// TIA Portal project "ProfiZumo" (V17)

(* hardware
DEVICE "S7-1500/ET200MP-Station_1"  S7-1500 station
   slot 0: "Profilschiene_0"  Rack  6ES7 590-1***0-0AA0
   slot 1: "PLC_1"  CPU 1516-3 PN/DP  6ES7 516-3AN01-0AB0  V2.9
      slot 3: "CPU-Display_1"  6ES7591-1BA00-0AA0
      slot 32768: "PROFINET-Schnittstelle_1"  X1
      slot 33024: "PROFINET-Schnittstelle_2"  X2
      slot 33280: "DP-Schnittstelle_1"  X3
      slot 34817: "Virtual CP interface port_1"  Virtual CP interface port  Virtual CP interface port
DEVICE "GSD-Geraet_1"  GSD.Device.PN
   slot 0: "Baugruppenträger"  Rack  V1.0
   slot 0: "profizumo"  Profizumo  123 444 555  V0.1.0
      slot 0: "Profizumo"  Profizumo
      slot 1: "X1"  X1
         slot 1: "X1 P1"  X1 P1
      slot 1: "unknown module_1"  unknown module  1.0
         slot 0: "unknown submodule"  unknown submodule
*)

// ===== PLC "PLC_1"  CPU 1516-3 PN/DP =====

VAR_GLOBAL   // PLC tag table "Standard-Variablentabelle"
   "leftMotor" AT %QD0 : UDInt;
END_VAR

DATA_BLOCK "States"   // DB3
{ S7_Optimized_Access := 'TRUE' }
VERSION : 0.1
   VAR
      leftMotorSetSpeed : UDInt;
   END_VAR
BEGIN
END_DATA_BLOCK

ORGANIZATION_BLOCK "Main"   // OB1, LAD, ProgramCycle
TITLE = "Main Program Sweep (Cycle)"
{ S7_Optimized_Access := 'TRUE' }
VERSION : 0.1
   VAR_INPUT
      Initial_Call : Bool;   // Initial call of this OB
      Remanence : Bool;   // =True, if remanent data are available
   END_VAR
   VAR_TEMP
      tempFloatIn : Real;
      tempIntIn : UDInt;
      tempFloatOut : Real;
   END_VAR
BEGIN

REGION Network 1
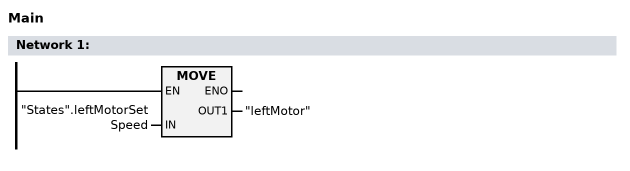
   RUNG wire#powerrail
      Move(in := "States".leftMotorSetSpeed, out1 => "leftMotor")
   END_RUNG
   // the same network as SCL:
   "leftMotor" := "States".leftMotorSetSpeed;
END_REGION
END_ORGANIZATION_BLOCK

ORGANIZATION_BLOCK "Counter"   // OB30, SCL, CyclicInterrupt
{ S7_Optimized_Access := 'TRUE' }
VERSION : 0.1
   VAR_INPUT
      Initial_Call : Bool;   // Initial call of this OB
      Event_Count : Int;   // Events discarded
   END_VAR
   VAR_TEMP
      tempLeftMotorSpeed : UDInt;
   END_VAR
BEGIN
   #tempLeftMotorSpeed:= "States".leftMotorSetSpeed + 1;
   IF #tempLeftMotorSpeed > 400 THEN
       #tempLeftMotorSpeed := 0;
   END_IF;
   "States".leftMotorSetSpeed := #tempLeftMotorSpeed;
END_ORGANIZATION_BLOCK